// TIA Portal V16 export
// export: Created 2022-03-28T07:44:08.625993Z, ExportSetting WithDefaults, DisplayName Totally Integrated Automation Portal, DisplayVersion V16 Update 5, DisplayName TIA Portal Version Control Interface, DisplayVersion V16 Update 2, DisplayName TIA Portal Openness, DisplayVersion V16 Update 5, DisplayName STEP 7 Professional, DisplayVersion V16 Update 5, DisplayName STEP 7 Safety, DisplayVersion V16, DisplayName WinCC Professional, DisplayVersion V16 Update 5
VAR_GLOBAL   // PLC tag table "Entradas PLC"
   "Rele Emergencia" AT %I0.0 : Bool;
   "Rele Barrera" AT %I0.1 : Bool;
   "Pulsador Rearme" AT %I0.2 : Bool;
   "Marcha 1" AT %I0.3 : Bool;
   "Marcha 2" AT %I0.4 : Bool;
   "Marcha 3" AT %I0.5 : Bool;
   Caudalímetro AT %I0.6 : Bool;
   Presostato AT %I0.7 : Bool;
   "Final Soldadura" AT %I1.1 : Bool;
   "Soldadura RDY" AT %I1.0 : Bool;
   "Acuse error soldadura" AT %I1.2 : Bool;
   "Fibra óptica Tornillo 1" AT %I1.3 : Bool;
   "Fibra óptica Tornillo 2" AT %I1.4 : Bool;
   "Cajón rechazo" AT %I1.5 : Bool;
   "Pinza 1 RE" AT %I2.0 : Bool;
   "Pinza 1 AV" AT %I2.1 : Bool;
   "Pinza 2 RE" AT %I2.2 : Bool;
   "Pinza 2 AV" AT %I2.3 : Bool;
   "Pinza 3 RE" AT %I2.4 : Bool;
   "Pinza 3 AV" AT %I2.5 : Bool;
   "Libre I 2.6" AT %I2.6 : Bool;
   "Libre I 2.7" AT %I2.7 : Bool;
   "Selector acuse pieza mala" AT %I3.0 : Bool;
   RobotOK AT %I3.1 : Bool;
   RobotNOK AT %I3.2 : Bool;
   RobotAuto AT %I3.3 : Bool;
   "Libre I 3.4" AT %I3.4 : Bool;
   "Libre I 3.5" AT %I3.5 : Bool;
   "Libre I 3.6" AT %I3.6 : Bool;
   "Libre I 3.7" AT %I3.7 : Bool;
   Tag_71 AT %IW64 : Word;
END_VAR
